// TIA Portal V21 export
DATA_BLOCK "PI"   // DB144
{ S7_Optimized_Access := 'TRUE' }
// stored: MemoryReserve 100
   VAR
      NOM1 : Real;
      SETPOINT : Real;
      "PID OUT" : Real;
      NOM2 : Real;
      "PID IN" : Real;
   END_VAR
   VAR RETAIN
      GAIN : Real;
      "TIME" : Real;
   END_VAR
   VAR
      NOM3 : Real;
   END_VAR
BEGIN
END_DATA_BLOCK
